TYPE WcStateBase :
STRUCT
	WcState AT %I* : BOOL;
END_STRUCT
END_TYPE

(* stored: Version 1.1.0.1, ProductVersion 3.1.4024.9
   DUT WcStateBase: Id {4ee7764e-3558-0b6b-0970-f4e41cb4cea7} *)
